Universal Robots PolyScope program: 180963.urp

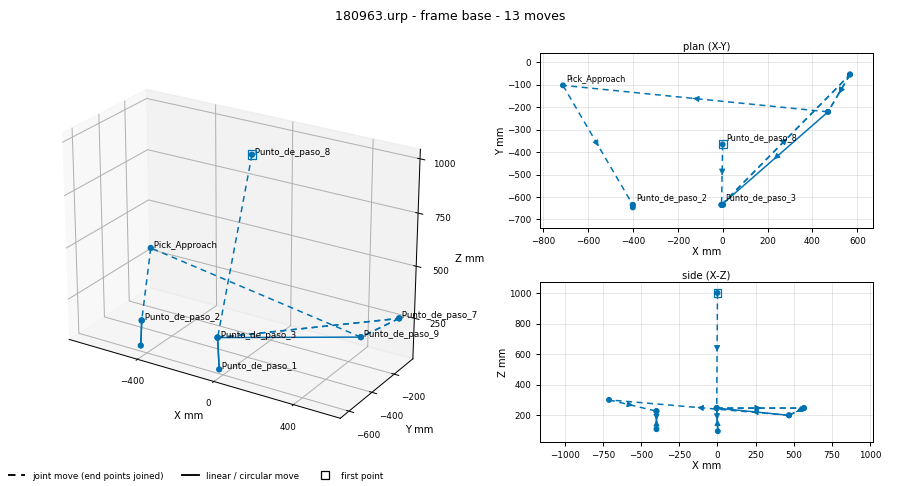
[picture p0: tool path of 180963.urp in frame base, 13 of 13 moves have a stored position in this frame; points joined in program order, loops and branches not executed]
Program 180963 (installation=default directory=/programs/usbdisk_2 createdIn=3.15.8.106339 lastSavedIn=3.15.8.106339 robotSerialNumber=2015350901)
Calibrated DH parameters: a=[0, -0.425, -0.39225, 0, 0, 0]; d=[0.089159, 0, 0, 0.10915, 0.09465, 0.0823]; alpha=[1.570796, 0, 0, 1.570796, -1.570796, 0]; deltaTheta=[0, 0, 0, 0, 0, 0]
Robot Program (runOnlyOnce=false)
  Set DigitalOutput pin=digital_out[4]; digitalValue=1
  Set NoAction (payload=0.92 tcpAsCog=true)
  MoveJ speed 60 deg/s, acceleration 80 deg/s^2 (useActiveTCP=true)
    Waypoint Punto_de_paso_8: TCP in base x=-0.02 y=-365.45 z=1001.059 mm, rx=0.0001 ry=2.2214 rz=-2.2214 rad; joints [-0.002, -90, 0.003, -89.997, 0.005, 0.001] deg; flange x=-0.028 y=-191.45 z=1001.059 mm, rx=0.0001 ry=2.2214 rz=-2.2214 rad
  Loop Counting (count=48) loopVariable(name=Bucle_1)
    Wait Sleep waitTime=0.5
    If digital_in[0]≟ True
      URCap Gripper (Robotiq_Grippers, Robotiq Inc.) dataModel(position=0.0, force=100.0, speed=100.0, positionInDouble=0.0, forceInDouble=100.0, speedInDouble=100.0, slaveIds=[9], blocking=true); state(isChildrenLocked=true)
      MoveJ speed 60 deg/s, acceleration 80 deg/s^2 (useActiveTCP=true)
        Waypoint Punto_de_paso_3: TCP in base x=-4.984 y=-634.851 z=245.361 mm, rx=2.2189 ry=2.1884 rz=0.0163 rad; joints [79.026, -71.339, 69.991, -88.968, -88.477, 79.825] deg; flange x=-9.341 y=-633.028 z=419.297 mm, rx=2.2189 ry=2.1884 rz=0.0163 rad
      MoveL speed 250 mm/s, acceleration 1200 mm/s^2 (useActiveTCP=true) feature=Base
        Waypoint Punto_de_paso_1: TCP in base x=2.281 y=-634.851 z=93.823 mm, rx=2.2189 ry=2.1884 rz=0.0163 rad; joints [79.682, -67.99, 87.92, -110.263, -88.48, 80.479] deg; flange x=-2.078 y=-633.028 z=267.759 mm, rx=2.2189 ry=2.1884 rz=0.0163 rad
      URCap Gripper (Robotiq_Grippers, Robotiq Inc.) dataModel(position=100.0, force=60.0, speed=0.0, positionInDouble=100.0, forceInDouble=60.0, speedInDouble=0.0, slaveIds=[9], blocking=true); state(isChildrenLocked=true)
      If digital_in[1]≟ True
        MoveL speed 250 mm/s, acceleration 1200 mm/s^2 (useActiveTCP=true) feature=Base
          Waypoint Punto_de_paso_6: TCP in base x=-4.985 y=-634.861 z=245.397 mm, rx=2.2189 ry=2.1882 rz=0.0162 rad; joints [79.024, -71.342, 69.991, -88.972, -88.474, 79.826] deg; flange x=-9.349 y=-633.018 z=419.333 mm, rx=2.2189 ry=2.1882 rz=0.0162 rad
        MoveJ speed 60 deg/s, acceleration 80 deg/s^2 (useActiveTCP=true)
          Waypoint Punto_de_paso_7: TCP in base x=567.496 y=-53.997 z=245.39 mm, rx=-0.0063 ry=3.1311 rz=0.0396 rad; joints [162.812, -80.424, 81.426, -91.128, -88.442, 72.584] deg; flange x=565.729 y=-58.402 z=419.325 mm, rx=-0.0063 ry=3.1311 rz=0.0396 rad
        Pallet pattern(dimensionality=Box firstAxisCount=3 secondAxisCount=2 thirdAxisCount=2 motionType=MoveL speed=0.25 acceleration=1.2 useActiveTCP=true, counterVariable(name=cont_2, initializeExpression=0), patternPoseVariable(name=pose_2), feature=Base, children(Waypoint(type=Fixed name=Esquina1_3, position(joints=3.210118532180786, -1.1934617201434534, 1.7991185188293457, -2.1883180777179163, -1.546206299458639, 1.6355385780334473 pose=0.567492969880056, 0.1546723281249082, 0.0058699773077803, -0.006151930623406608, 3.1311351141521486, 0.03965077849473769), poseInFeatureCoordinates=[0.567493, 0.154672, 0.00587, -0.006152, 3.131135, 0.039651], outputFlangePose=[0.565727, 0.150263, 0.179805, -0.006152, 3.131135, 0.039651]), Waypoint(type=Fixed name=Esquina2_3, position(joints=2.722168445587158, -1.2027457396136683, 1.8092279434204102, -2.17611533800234, -1.5436065832721155, 1.1472989320755005 pose=0.5674808646938327, -0.12589184612829943, 0.00580690033982173, -0.006352381332958704, 3.131274375057311, 0.03959162558746121), poseInFeatureCoordinates=[0.567481, -0.125892, 0.005807, -0.006352, 3.131274, 0.039592], outputFlangePose=[0.565739, -0.130295, 0.179742, -0.006352, 3.131274, 0.039592]), Waypoint(type=Fixed name=Esquina3_3, position(joints=2.7693684101104736, -1.0548537413226526, 1.5803771018981934, -2.0966489950763147, -1.5434873739825647, 1.1945942640304565 pose=0.6418902038367187, -0.12592260538511021, 0.005884267349809402, -0.0062344177154403276, 3.1310471864331455, 0.03960822596585996), poseInFeatureCoordinates=[0.64189, -0.125923, 0.005884, -0.006234, 3.131047, 0.039608], outputFlangePose=[0.640109, -0.130328, 0.179819, -0.006234, 3.131047, 0.039608]), Waypoint(type=Fixed name=Esquina4_3, position(joints=3.2053704261779785, -1.0456422011004847, 1.5686016082763672, -2.105522934590475, -1.5461705366717737, 1.6307384967803955 pose=0.6418728923902715, 0.1566889947437647, 0.00589026099160575, -0.006231708048624386, 3.131114325923235, 0.03962024847271563), poseInFeatureCoordinates=[0.641873, 0.156689, 0.00589, -0.006232, 3.131114, 0.03962], outputFlangePose=[0.640103, 0.152283, 0.179825, -0.006232, 3.131114, 0.03962]), Waypoint(type=Fixed name=Esquina5_3, position(joints=3.210106611251831, -1.2432940641986292, 1.753187656402588, -2.0926736036883753, -1.5463264624225062, 1.6353471279144287 pose=0.567526646379355, 0.15463688657500974, 0.04504798397595455, -0.006433893391734468, 3.1310077605775994, 0.039472178897731205), poseInFeatureCoordinates=[0.567527, 0.154637, 0.045048, -0.006434, 3.131008, 0.039472], outputFlangePose=[0.565739, 0.150247, 0.218983, -0.006434, 3.131008, 0.039472]), Waypoint(type=Fixed name=Esquina6_3, position(joints=2.7221803665161133, -1.2527697722064417, 1.7629132270812988, -2.079860035573141, -1.5436185042010706, 1.1472629308700562 pose=0.5674930746245486, -0.12589320014777475, 0.04500306731764181, -0.006429051227423877, 3.1312035508516614, 0.03952006184790415), poseInFeatureCoordinates=[0.567493, -0.125893, 0.045003, -0.006429, 3.131204, 0.03952], outputFlangePose=[0.565739, -0.130288, 0.218939, -0.006429, 3.131204, 0.03952]), Waypoint(type=Fixed name=Esquina7_3, position(joints=2.769392251968384, -1.097630802785055, 1.5351715087890625, -2.0083535353290003, -1.5434630552874964, 1.1945703029632568 pose=0.6417999498946394, -0.12586420612784946, 0.045060158559726754, -0.006303130183906217, 3.131326550755029, 0.039826230196334876), poseInFeatureCoordinates=[0.6418, -0.125864, 0.04506, -0.006303, 3.131327, 0.039826], outputFlangePose=[0.640068, -0.130293, 0.218995, -0.006303, 3.131327, 0.039826]), Waypoint(type=Fixed name=Esquina8_3, position(joints=3.2053825855255127, -1.0881555716144007, 1.5237679481506348, -2.018078152333395, -1.5462663809405726, 1.6307024955749512 pose=0.6418211706335804, 0.15666900987310411, 0.04499527063606923, -0.0063045339491769855, 3.1312075114374385, 0.039461988946448666), poseInFeatureCoordinates=[0.641821, 0.156669, 0.044995, -0.006305, 3.131208, 0.039462], outputFlangePose=[0.640068, 0.152281, 0.218931, -0.006305, 3.131208, 0.039462]))); actionSequence(name=SecuenciaPalé motionType=MoveL speed=0.25 acceleration=1.2 useActiveTCP=true, anchorWaypoint(type=Fixed name=PuntoDePatrón_3, position(joints=3.2101783752441406, -1.1934259573565882, 1.799178123474121, -2.1882460753070276, -1.5462544600116175, 1.6356104612350464 pose=0.5674348168928285, 0.15469056063082479, 0.005816975097799659, -0.006129744092453944, 3.131301743890378, 0.03956122754647195), poseInFeatureCoordinates=[0.567435, 0.154691, 0.005817, -0.00613, 3.131302, 0.039561], outputFlangePose=[0.565698, 0.150291, 0.179753, -0.00613, 3.131302, 0.039561]), feature=Base, children(Waypoint(type=Fixed name=Acercar_3, position(joints=3.2101664543151855, -1.2652280966388147, 1.7269015312194824, -2.04431659380068, -1.5462544600116175, 1.6355984210968018 pose=0.5674529789399674, 0.1546849170285572, 0.06466123293220949, -0.006132505776048727, 3.1311523459374597, 0.03957472334820667), poseInFeatureCoordinates=[0.567453, 0.154685, 0.064661, -0.006133, 3.131152, 0.039575], outputFlangePose=[0.56569, 0.150284, 0.238597, -0.006133, 3.131152, 0.039575]), Waypoint=PuntoDePatrón_3, Contributed(strategyProgramNodeType=Gripper strategyURCapDeveloper=Robotiq Inc. strategyURCapName=Robotiq_Grippers, dataModel(position=46.27450980392157, force=0.0, speed=0.0, positionInDouble=46.27450980392157, forceInDouble=0.0, speedInDouble=0.0, slaveIds=[9], blocking=true), state(isChildrenLocked=true)), Set(type=NoAction payload=0.92 tcpAsCog=true), Wait(type=Sleep, waitTime=0.5), Waypoint(type=Fixed name=Salir_3, position(joints=3.210106611251831, -1.336862866078512, 1.5819954872131348, -1.8278430143939417, -1.546218220387594, 1.635562539100647 pose=0.5674802178683294, 0.15466149992245093, 0.15231295173423248, -0.006096492881740091, 3.1310857525030147, 0.0396367444149853), poseInFeatureCoordinates=[0.56748, 0.154661, 0.152313, -0.006096, 3.131086, 0.039637], outputFlangePose=[0.565705, 0.150253, 0.326248, -0.006096, 3.131086, 0.039637])))
          Pattern -> pattern
          AnchoredSequence -> SecuenciaPalé
        MoveJ speed 60 deg/s, acceleration 80 deg/s^2 (useActiveTCP=true)
          Waypoint Punto_de_paso_9: TCP in base x=469.429 y=-220.494 z=198.064 mm, rx=-0.006 ry=3.1313 rz=0.0395 rad; joints [141.936, -86.63, 95.196, -98.126, -88.508, 51.71] deg; flange x=467.689 y=-224.886 z=372 mm, rx=-0.006 ry=3.1313 rz=0.0395 rad
      Else 
        MoveL speed 250 mm/s, acceleration 1200 mm/s^2 (useActiveTCP=true) feature=Base
          Waypoint Punto_de_paso_6: TCP in base x=-4.985 y=-634.861 z=245.397 mm, rx=2.2189 ry=2.1882 rz=0.0162 rad; joints [79.024, -71.342, 69.991, -88.972, -88.474, 79.826] deg; flange x=-9.349 y=-633.018 z=419.333 mm, rx=2.2189 ry=2.1882 rz=0.0162 rad
        MoveJ speed 60 deg/s, acceleration 80 deg/s^2 (useActiveTCP=true)
          Waypoint Punto_de_paso_7: TCP in base x=567.496 y=-53.997 z=245.39 mm, rx=-0.0063 ry=3.1311 rz=0.0396 rad; joints [162.812, -80.424, 81.426, -91.128, -88.442, 72.584] deg; flange x=565.729 y=-58.402 z=419.325 mm, rx=-0.0063 ry=3.1311 rz=0.0396 rad
        Pallet pattern(dimensionality=Box firstAxisCount=3 secondAxisCount=2 thirdAxisCount=2 motionType=MoveL speed=0.25 acceleration=1.2 useActiveTCP=true, counterVariable(name=cont_3, initializeExpression=0), patternPoseVariable(name=pose_3), feature=Base, children(Waypoint(type=Fixed name=Esquina1_2, position(joints=3.192996025085449, -0.7955716292010706, 1.138380527496338, -1.9248436133014124, -1.5460384527789515, 1.6184449195861816 pose=0.7574537820699964, 0.15461755712088196, 0.005731016151258234, -0.00609657689336091, 3.1313383556234093, 0.039588255529352745), poseInFeatureCoordinates=[0.757454, 0.154618, 0.005731, -0.006097, 3.131338, 0.039588], outputFlangePose=[0.755723, 0.150215, 0.179667, -0.006097, 3.131338, 0.039588]), Waypoint(type=Fixed name=Esquina2_2, position(joints=2.825104236602783, -0.8036816755877894, 1.1502723693847656, -1.9193227926837366, -1.5435588995562952, 1.2507007122039795 pose=0.7574916638142584, -0.1258768062285422, 0.005857519520291676, -0.005688303076922408, 3.1309757121132145, 0.03955232911095843), poseInFeatureCoordinates=[0.757492, -0.125877, 0.005858, -0.005688, 3.130976, 0.039552], outputFlangePose=[0.755697, -0.130275, 0.179793, -0.005688, 3.130976, 0.039552]), Waypoint(type=Fixed name=Esquina3_2, position(joints=2.852973699569702, -0.597450081502096, 0.767547607421875, -1.7429693380938929, -1.5435469786273401, 1.2776325941085815 pose=0.8317430966481256, -0.12580841114680763, 0.005829509205152461, -0.007160338788195467, 3.1315265422807346, 0.03994416308442988), poseInFeatureCoordinates=[0.831743, -0.125808, 0.00583, -0.00716, 3.131527, 0.039944], outputFlangePose=[0.830048, -0.13025, 0.179765, -0.00716, 3.131527, 0.039944]), Waypoint(type=Fixed name=Esquina4_2, position(joints=3.190742015838623, -0.5867527166949671, 0.7490091323852539, -1.7446344534503382, -1.5461466948138636, 1.6160271167755127 pose=0.8319391801105738, 0.1565289028054177, 0.005989460838711269, -0.006357874558818689, 3.130933086022148, 0.03940253366037798), poseInFeatureCoordinates=[0.831939, 0.156529, 0.005989, -0.006358, 3.130933, 0.039403], outputFlangePose=[0.830138, 0.152147, 0.179925, -0.006358, 3.130933, 0.039403]), Waypoint(type=Fixed name=Esquina5_2, position(joints=3.1928043365478516, -0.8262260595904749, 1.087986946105957, -1.8442395369159144, -1.5461586157428187, 1.618432879447937 pose=0.7576159535703009, 0.15444832418425353, 0.04508894519120757, -0.005821976001198541, 3.1308889916076055, 0.03942740020590309), poseInFeatureCoordinates=[0.757616, 0.154448, 0.045089, -0.005822, 3.130889, 0.039427], outputFlangePose=[0.755806, 0.150063, 0.219024, -0.005822, 3.130889, 0.039427]), Waypoint(type=Fixed name=Esquina6_2, position(joints=2.825200319290161, -0.8346231619464319, 1.1000456809997559, -1.8379634062396448, -1.54352313676943, 1.2507367134094238 pose=0.7574430275191568, -0.12577450110331873, 0.04516948076039001, -0.005778645966655003, 3.131145737676816, 0.03970240185928713), poseInFeatureCoordinates=[0.757443, -0.125775, 0.045169, -0.005779, 3.131146, 0.039702], outputFlangePose=[0.755678, -0.13019, 0.219105, -0.005779, 3.131146, 0.039702]), Waypoint(type=Fixed name=Esquina7_2, position(joints=2.852961778640747, -0.6148923079120081, 0.6999130249023438, -1.6578500906573694, -1.5435469786273401, 1.2787704467773438 pose=0.8317510460533852, -0.12582113196370007, 0.0450078807172227, -0.00535925258441192, 3.1315848064555354, 0.03997251863631863), poseInFeatureCoordinates=[0.831751, -0.125821, 0.045008, -0.005359, 3.131585, 0.039973], outputFlangePose=[0.830063, -0.130265, 0.218943, -0.005359, 3.131585, 0.039973]), Waypoint(type=Fixed name=Esquina8_2, position(joints=3.1906464099884033, -0.603487793599264, 0.6807408332824707, -1.6593955198871058, -1.54608661333193, 1.616015076637268 pose=0.8318883312292512, 0.15646154575255128, 0.04495024458881555, -0.006223512297969529, 3.1311691424662915, 0.03948121941613682), poseInFeatureCoordinates=[0.831888, 0.156462, 0.04495, -0.006224, 3.131169, 0.039481], outputFlangePose=[0.830128, 0.152071, 0.218886, -0.006224, 3.131169, 0.039481]))); actionSequence(name=SecuenciaPalé motionType=MoveL speed=0.25 acceleration=1.2 useActiveTCP=true, anchorWaypoint(type=Fixed name=PuntoDePatrón_2, position(joints=3.193079948425293, -0.7957037130938929, 1.138512134552002, -1.92503530183901, -1.5461104551898401, 1.6185647249221802 pose=0.7574507383068799, 0.15466316354350226, 0.005788766889687408, -0.0060431079313838796, 3.1311467721576096, 0.03948974769580263), poseInFeatureCoordinates=[0.757451, 0.154663, 0.005789, -0.006043, 3.131147, 0.03949], outputFlangePose=[0.755686, 0.150272, 0.179724, -0.006043, 3.131147, 0.03949]), feature=Base, children(Waypoint(type=Fixed name=Acercar_2, position(joints=3.1930320262908936, -0.8430803457843226, 1.046501636505127, -1.785705868397848, -1.5461104551898401, 1.618432879447937 pose=0.757496438799957, 0.15462883605415753, 0.07214412968039591, -0.00617549290963571, 3.131086591061233, 0.039492030587168735), poseInFeatureCoordinates=[0.757496, 0.154629, 0.072144, -0.006175, 3.131087, 0.039492], outputFlangePose=[0.755722, 0.150237, 0.24608, -0.006175, 3.131087, 0.039492]), Waypoint=PuntoDePatrón_2, Contributed(strategyProgramNodeType=Gripper strategyURCapDeveloper=Robotiq Inc. strategyURCapName=Robotiq_Grippers, dataModel(position=46.27450980392157, force=0.0, speed=0.0, positionInDouble=46.27450980392157, forceInDouble=0.0, speedInDouble=0.0, slaveIds=[9], blocking=true), state(isChildrenLocked=true)), Set(type=NoAction payload=0.92 tcpAsCog=true), Wait(type=Sleep, waitTime=0.5), Waypoint(type=Fixed name=Salir_2, position(joints=3.1930079460144043, -0.8377855459796351, 1.061448574066162, -1.8056963125811976, -1.5461824576007288, 1.618492841720581 pose=0.7574308055292409, 0.15458855312723221, 0.06285855546539276, -0.006038912122477081, 3.131336344477635, 0.039363364445480616), poseInFeatureCoordinates=[0.757431, 0.154589, 0.062859, -0.006039, 3.131336, 0.039363], outputFlangePose=[0.755699, 0.150211, 0.236795, -0.006039, 3.131336, 0.039363])))
          Pattern -> pattern
          AnchoredSequence -> SecuenciaPalé
        MoveJ speed 60 deg/s, acceleration 80 deg/s^2 (useActiveTCP=true)
          Waypoint Punto_de_paso_9: TCP in base x=469.429 y=-220.494 z=198.064 mm, rx=-0.006 ry=3.1313 rz=0.0395 rad; joints [141.936, -86.63, 95.196, -98.126, -88.508, 51.71] deg; flange x=467.689 y=-224.886 z=372 mm, rx=-0.006 ry=3.1313 rz=0.0395 rad
    Else 
      MoveJ speed 60 deg/s, acceleration 80 deg/s^2 (useActiveTCP=true)
        Waypoint Pick_Approach: TCP in base x=-711.456 y=-102.481 z=299.284 mm, rx=-2.2313 ry=-2.2052 rz=0.0194 rad; joints [-0.655, -56.149, 39.509, -74.037, -89.673, 0.019] deg; flange x=-709.387 y=-101.512 z=473.269 mm, rx=-2.2313 ry=-2.2052 rz=0.0194 rad
      Set DigitalOutput pin=digital_out[0]; digitalValue=1
      URCap Gripper (Robotiq_Grippers, Robotiq Inc.) dataModel(position=0.0, force=100.0, speed=100.0, positionInDouble=0.0, forceInDouble=100.0, speedInDouble=100.0, slaveIds=[9], blocking=true); state(isChildrenLocked=true)
      Pallet pattern(dimensionality=Box firstAxisCount=3 secondAxisCount=4 thirdAxisCount=2 motionType=MoveL speed=0.25 acceleration=1.2 useActiveTCP=true, counterVariable(name=cont_1, initializeExpression=0), patternPoseVariable(name=pose_1), feature=Base, children(Waypoint(type=Fixed name=Esquina1_1, position(joints=-0.18097383180727178, -0.8358929792987269, 1.0883221626281738, -1.7965696493731897, -1.5651000181781214, -0.16705257097353154 pose=-0.7601915562013655, 0.0266503171122866, 0.04777000130510595, 2.2190327993823185, 2.1881879520421847, 0.016574802257979485), poseInFeatureCoordinates=[-0.760192, 0.02665, 0.04777, 2.219033, 2.188188, 0.016575], outputFlangePose=[-0.764575, 0.02846, 0.221705, 2.219033, 2.188188, 0.016575]), Waypoint(type=Fixed name=Esquina2_1, position(joints=0.18237368762493134, -0.7247164885150355, 0.8902912139892578, -1.713909927998678, -1.556030575429098, 0.19614169001579285 pose=-0.7602989700536434, -0.2550553421360529, 0.04791783807894495, 2.2191561251364678, 2.1884482009752726, 0.016046654291889565), poseInFeatureCoordinates=[-0.760299, -0.255055, 0.047918, 2.219156, 2.188448, 0.016047], outputFlangePose=[-0.764608, -0.253237, 0.221855, 2.219156, 2.188448, 0.016047]), Waypoint(type=Fixed name=Esquina3_1, position(joints=0.2439100742340088, -1.1804049650775355, 1.646017074584961, -2.0147369543658655, -1.5547125975238245, 0.2575424909591675 pose=-0.5561492610342607, -0.25513311833082325, 0.04781594728015798, 2.2189789391088226, 2.188551714403257, 0.01628750845827454), poseInFeatureCoordinates=[-0.556149, -0.255133, 0.047816, 2.218979, 2.188552, 0.016288], outputFlangePose=[-0.560484, -0.253328, 0.221753, 2.218979, 2.188552, 0.016288]), Waypoint(type=Fixed name=Esquina4_1, position(joints=-0.2470000425921839, -1.2951515356646937, 1.8051743507385254, -2.0541847387896937, -1.5668371359454554, -0.233161751423971 pose=-0.5561619398584727, 0.026622709814255765, 0.04789213782483884, 2.219111383268741, 2.1884977975693087, 0.016255022477246594), poseInFeatureCoordinates=[-0.556162, 0.026623, 0.047892, 2.219111, 2.188498, 0.016255], outputFlangePose=[-0.560487, 0.028424, 0.221829, 2.219111, 2.188498, 0.016255]), Waypoint(type=Fixed name=Esquina5_1, position(joints=-0.18093759218324834, -0.8012259642230433, 1.14683198928833, -1.8897164503680628, -1.5651000181781214, -0.1671364943133753 pose=-0.7601796041274209, 0.02662040496544379, 0.002786680283432208, 2.21888362687355, 2.1883036285782294, 0.016600609766856882), poseInFeatureCoordinates=[-0.76018, 0.02662, 0.002787, 2.218884, 2.188304, 0.016601], outputFlangePose=[-0.764568, 0.028431, 0.176722, 2.218884, 2.188304, 0.016601]), Waypoint(type=Fixed name=Esquina6_1, position(joints=0.18232575058937073, -0.6965535322772425, 0.9561986923217773, -1.8076613585101526, -1.5561144987689417, 0.19618962705135345 pose=-0.7602578289724236, -0.25498718622155864, 0.0027624210599998256, 2.2191826900240716, 2.1882615070335847, 0.01653091843965047), poseInFeatureCoordinates=[-0.760258, -0.254987, 0.002762, 2.219183, 2.188262, 0.016531], outputFlangePose=[-0.764618, -0.253194, 0.176699, 2.219183, 2.188262, 0.016531]), Waypoint(type=Fixed name=Esquina7_1, position(joints=0.24382618069648743, -1.1275656859027308, 1.6988763809204102, -2.120336357747213, -1.5546887556659144, 0.25755447149276733 pose=-0.556140284400231, -0.25508519871568325, 0.002721845055412203, 2.219033733002505, 2.1883936023677637, 0.01639980187738091), poseInFeatureCoordinates=[-0.55614, -0.255085, 0.002722, 2.219034, 2.188394, 0.0164], outputFlangePose=[-0.560492, -0.25328, 0.176658, 2.219034, 2.188394, 0.0164]), Waypoint(type=Fixed name=Esquina8_1, position(joints=-0.24702388445009404, -1.2361066977130335, 1.8596925735473633, -2.1674936453448694, -1.5668614546405237, -0.23302966753114873 pose=-0.5561212285069219, 0.02663229146008206, 0.0027723210496512773, 2.2191359646675024, 2.1881804005323966, 0.016493918892521373), poseInFeatureCoordinates=[-0.556121, 0.026632, 0.002772, 2.219136, 2.18818, 0.016494], outputFlangePose=[-0.56049, 0.02844, 0.176708, 2.219136, 2.18818, 0.016494]))); actionSequence(name=SecuenciaPalé motionType=MoveL speed=0.25 acceleration=1.2 useActiveTCP=true, anchorWaypoint(type=Fixed name=PuntoDePatrón_1, position(joints=-0.18111783662904912, -0.833592716847555, 1.0937647819519043, -1.8043072859393519, -1.5651238600360315, -0.16750842729677373 pose=-0.760140621841317, 0.0267573771675379, 0.04417524102855655, 2.218695566768652, 2.188538527762078, 0.016598222081218517), poseInFeatureCoordinates=[-0.760141, 0.026757, 0.044175, 2.218696, 2.188539, 0.016598], outputFlangePose=[-0.764525, 0.028564, 0.218111, 2.218696, 2.188539, 0.016598]), feature=Base, children(Waypoint(type=Fixed name=Acercar_1, position(joints=-0.18091375032533819, -0.8725007216082972, 0.9320721626281738, -1.6038840452777308, -1.5651000181781214, -0.16700488725771123 pose=-0.7602410893304963, 0.02661341127016694, 0.13261767110748715, 2.2191200353843263, 2.1883021811544228, 0.01642365577434757), poseInFeatureCoordinates=[-0.760241, 0.026613, 0.132618, 2.21912, 2.188302, 0.016424], outputFlangePose=[-0.764595, 0.028417, 0.306554, 2.21912, 2.188302, 0.016424]), Waypoint=PuntoDePatrón_1, Set(type=NoAction payload=1.17 tcpAsCog=true), Contributed(strategyProgramNodeType=Gripper strategyURCapDeveloper=Robotiq Inc. strategyURCapName=Robotiq_Grippers, dataModel(position=100.0, force=60.0, speed=20.0, positionInDouble=100.0, forceInDouble=60.0, speedInDouble=20.0, slaveIds=[9], blocking=true), state(isChildrenLocked=true)), Wait(type=Sleep, waitTime=0.5), Waypoint(type=Fixed name=Salir_1, position(joints=-0.18088990846742803, -0.8725245634662073, 0.932096004486084, -1.6038840452777308, -1.5650399366961878, -0.16698104539980108 pose=-0.7602368616701288, 0.026578742460800883, 0.13262427366672808, 2.2190968118115975, 2.1882775388370828, 0.01634774400074541), poseInFeatureCoordinates=[-0.760237, 0.026579, 0.132624, 2.219097, 2.188278, 0.016348], outputFlangePose=[-0.764589, 0.028393, 0.30656, 2.219097, 2.188278, 0.016348])))
        Pattern -> pattern
        AnchoredSequence -> SecuenciaPalé
      MoveJ speed 60 deg/s, acceleration 80 deg/s^2 (useActiveTCP=true)
        Waypoint Punto_de_paso_2: TCP in base x=-400.404 y=-634.867 z=225.48 mm, rx=2.2192 ry=2.1881 rz=0.0163 rad; joints [48.89, -52.074, 43.558, -80.995, -88.525, 49.693] deg; flange x=-404.755 y=-633.039 z=399.416 mm, rx=2.2192 ry=2.1881 rz=0.0163 rad
      MoveL speed 250 mm/s, acceleration 1200 mm/s^2 (useActiveTCP=true) feature=Base
        Waypoint Punto_de_paso_4: TCP in base x=-400.216 y=-646.147 z=107.058 mm, rx=2.2191 ry=2.1883 rz=0.0166 rad; joints [49.467, -50.54, 58.338, -97.309, -88.525, 50.262] deg; flange x=-404.586 y=-644.363 z=280.994 mm, rx=2.2191 ry=2.1883 rz=0.0166 rad
        URCap Gripper (Robotiq_Grippers, Robotiq Inc.) dataModel(position=0.0, force=60.0, speed=0.0, positionInDouble=0.0, forceInDouble=60.0, speedInDouble=0.0, slaveIds=[9], blocking=true); state(isChildrenLocked=true)
      MoveL speed 250 mm/s, acceleration 1200 mm/s^2 (useActiveTCP=true) feature=Base
        Waypoint Punto_de_paso_5: TCP in base x=-400.441 y=-634.851 z=225.43 mm, rx=2.2193 ry=2.188 rz=0.0164 rad; joints [48.886, -52.07, 43.557, -80.993, -88.523, 49.693] deg; flange x=-404.805 y=-633.031 z=399.366 mm, rx=2.2193 ry=2.188 rz=0.0164 rad
  Set DigitalOutput pin=digital_out[4]; digitalValue=0
  Popup Warning (haltProgram=true message=Pallet terminado. Recolectar Pallets en  Packaging Area y cargar mas  cubos. inputType=Text)
Event  expression=digital_in[0]≟ True
  Wait Sleep waitTime=1
  Set DigitalOutput pin=digital_out[4]; digitalValue=0
Event  expression=digital_in[0]≟ False
  Set DigitalOutput pin=digital_out[4]; digitalValue=1
